INTERFACE IByteList EXTENDS IReadOnlyByteList

METHOD Set
VAR_INPUT
	index : DINT;
	value : BYTE;
END_VAR
END_METHOD

END_INTERFACE

(* stored: Version 1.1.0.1
   Itf IByteList: Id {518eb55c-df07-0206-0227-e692a273d945}
   Method Set: Id {267c54d8-2df6-0ce5-162c-03537dc39a04} *)
